ABB RobotStudio station: 101229220_Individual_Assignment_RSD.rspag

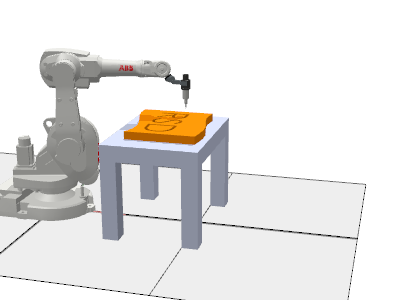
--- station ---
Station Project2 (saved by RobotStudio 24.1.10713.1)
Controller IRB1600_6_120
  mechanical unit ROB_1: IRB1600_6_120__02, 6 joints, base frame (0, 0, 0) mm
Layout (positions relative to the parent item):
  - IRB1600_6_120__02 [mechanism, from %ABB.RobotStudio.Models.IRB1600%\IRB1600_6_120_G_03.rslib] at (0, 0, 0) mm; joint values [0.2858, -0.0359, 0.0676, -0.2293, 0.9102, 0.378] (rad or m)
  - MyTool [mechanism, from Training Objects\myTool.rslib] at (742.97, 206.13, 890.95) mm, rotated rx -180 ry 38 rz 179.42 deg
  - Table [part] at (800, 0, 0) mm, rotated rx 0 ry 0 rz 90 deg, size 800 x 600 x 600 mm
  - RSD_Flag_3 [part] at (840.17, 31.01, 600) mm, rotated rx 0 ry 0 rz -90 deg, size 540.6 x 505.2 x 50 mm
Attachment: MyTool is attached to IRB1600_6_120__02 / Link6
Attachment: RSD_Flag_3 is attached to Table
Targets, tools, work objects and paths stored in the station and not in the controller backup, written as RAPID:
! task T_ROB1
MODULE Module1
  CONST robtarget Target_1090:=[[359.518,326.698,50],[0,0,1,0],[-1,0,-1,0],[9E+09,9E+09,9E+09,9E+09,9E+09,9E+09]];
  CONST robtarget Target_1100:=[[359.518,326.698,50],[0,0,1,0],[0,0,-1,0],[9E+09,9E+09,9E+09,9E+09,9E+09,9E+09]];
  CONST robtarget Target_1110:=[[359.518,326.698,50],[0,0,1,0],[0,0,-1,0],[9E+09,9E+09,9E+09,9E+09,9E+09,9E+09]];
  CONST robtarget Target_1120:=[[359.518,326.698,50],[0,0,1,0],[0,0,0,0],[9E+09,9E+09,9E+09,9E+09,9E+09,9E+09]];
  CONST robtarget Target_150_2:=[[193.305,628.255,70],[0,0,1,0],[0,0,0,0],[9E+09,9E+09,9E+09,9E+09,9E+09,9E+09]];
  CONST robtarget Target_310_2:=[[193.305,628.255,70],[0,0,1,0],[0,0,0,0],[9E+09,9E+09,9E+09,9E+09,9E+09,9E+09]];
  CONST robtarget Target_410_2:=[[359.518,611.634,70],[0,0,1,0],[0,0,0,0],[9E+09,9E+09,9E+09,9E+09,9E+09,9E+09]];
  CONST robtarget Target_930_2:=[[378.513525558,343.318900025,50],[0,0,1,0],[0,0,0,0],[9E+09,9E+09,9E+09,9E+09,9E+09,9E+09]];
  CONST robtarget Target_1130:=[[212.30091872,326.697639341,50],[0,1,0,0],[0,0,0,0],[9E+09,9E+09,9E+09,9E+09,9E+09,9E+09]];
  CONST robtarget Target_1140:=[[359.517799062,326.697639341,50],[0,1,0,0],[0,0,0,0],[9E+09,9E+09,9E+09,9E+09,9E+09,9E+09]];
  CONST robtarget Target_1150:=[[356.586817826,266.779478617,50],[0,-0.64587981,0.763439107,0],[0,0,0,0],[9E+09,9E+09,9E+09,9E+09,9E+09,9E+09]];
  CONST robtarget Target_1160:=[[347.459964861,240.920061884,50],[0,-0.495864219,0.868400067,0],[0,0,0,0],[9E+09,9E+09,9E+09,9E+09,9E+09,9E+09]];
  CONST robtarget Target_1170:=[[333.176068961,224.261700172,50],[0,-0.337129953,0.941458122,0],[0,0,0,0],[9E+09,9E+09,9E+09,9E+09,9E+09,9E+09]];
  CONST robtarget Target_1180:=[[313.586726012,213.020088593,50],[0,-0.178855224,0.983875403,0],[0,0,0,0],[9E+09,9E+09,9E+09,9E+09,9E+09,9E+09]];
  CONST robtarget Target_1190:=[[296.334747847,208.790571366,50],[0,-0.066549315,0.997783137,0],[0,0,0,0],[9E+09,9E+09,9E+09,9E+09,9E+09,9E+09]];
  CONST robtarget Target_1200:=[[265.874803603,209.643895017,50],[0,0.098590622,0.995128077,0],[0,0,0,0],[9E+09,9E+09,9E+09,9E+09,9E+09,9E+09]];
  CONST robtarget Target_1210:=[[245.580541116,217.101201708,50],[0,0.253457957,0.967346403,0],[0,0,0,0],[9E+09,9E+09,9E+09,9E+09,9E+09,9E+09]];
  CONST robtarget Target_1220:=[[229.552896885,230.049460588,50],[0,0.410722051,0.911760603,0],[0,0,0,0],[9E+09,9E+09,9E+09,9E+09,9E+09,9E+09]];
  CONST robtarget Target_1230:=[[221.019660374,242.663810214,50],[0,0.524154537,0.851623169,0],[0,0,0,0],[9E+09,9E+09,9E+09,9E+09,9E+09,9E+09]];
  CONST robtarget Target_1240:=[[214.155970136,266.853680674,50],[0,0.663168665,0.748469987,0],[0,0,0,0],[9E+09,9E+09,9E+09,9E+09,9E+09,9E+09]];
  CONST robtarget Target_1250:=[[212.30091872,326.697639341,50],[0,0.707106781,0.707106781,0],[0,0,0,0],[9E+09,9E+09,9E+09,9E+09,9E+09,9E+09]];
  CONST robtarget Target_1260:=[[297.781687951,611.633536777,50],[0,1,0,0],[0,0,0,0],[9E+09,9E+09,9E+09,9E+09,9E+09,9E+09]];
  CONST robtarget Target_1270:=[[359.517799062,611.633536777,50],[0,1,0,0],[0,0,0,0],[9E+09,9E+09,9E+09,9E+09,9E+09,9E+09]];
  CONST robtarget Target_1280:=[[297.781687951,611.633536777,50],[0,1,0,0],[0,0,0,0],[9E+09,9E+09,9E+09,9E+09,9E+09,9E+09]];
  CONST robtarget Target_120_2:=[[522.92,479.312,50],[0,-0.111729096,0.993738703,0],[0,0,-1,0],[9E+09,9E+09,9E+09,9E+09,9E+09,9E+09]];
  PROC Path_1()
    MoveL Target_140,v1500,fine,MyTool\WObj:=Table_Workobject;
    MoveL Target_130,v1500,fine,MyTool\WObj:=Table_Workobject;
    MoveC Target_120,Target_110,v1500,fine,MyTool\WObj:=Table_Workobject;
    MoveC Target_100,Target_90,v1500,fine,MyTool\WObj:=Table_Workobject;
    MoveL Target_80,v1500,fine,MyTool\WObj:=Table_Workobject;
    MoveC Target_70,Target_60,v1500,fine,MyTool\WObj:=Table_Workobject;
    MoveC Target_50,Target_40,v1500,fine,MyTool\WObj:=Table_Workobject;
    MoveC Target_30,Target_20,v1500,fine,MyTool\WObj:=Table_Workobject;
    MoveL Target_10,v1500,fine,MyTool\WObj:=Table_Workobject;
    MoveL Target_140_2,v1500,fine,MyTool\WObj:=Table_Workobject;
  ENDPROC
  PROC Path_2()
    MoveL Target_160,v1500,fine,MyTool\WObj:=Table_Workobject;
    MoveL Target_170,v1500,fine,MyTool\WObj:=Table_Workobject;
    MoveC Target_180,Target_190,v150,fine,MyTool\WObj:=Table_Workobject;
    MoveC Target_200,Target_210,v150,fine,MyTool\WObj:=Table_Workobject;
    MoveC Target_220,Target_230,v150,fine,MyTool\WObj:=Table_Workobject;
    MoveC Target_240,Target_250,v150,fine,MyTool\WObj:=Table_Workobject;
    MoveL Target_260,v1500,fine,MyTool\WObj:=Table_Workobject;
    MoveL Target_270,v1500,fine,MyTool\WObj:=Table_Workobject;
    MoveL Target_280,v1500,fine,MyTool\WObj:=Table_Workobject;
    MoveL Target_290,v1500,fine,MyTool\WObj:=Table_Workobject;
    MoveL Target_300,v1500,fine,MyTool\WObj:=Table_Workobject;
    MoveL Target_310,v1500,fine,MyTool\WObj:=Table_Workobject;
    MoveL Target_150,v1500,fine,MyTool\WObj:=Table_Workobject;
    MoveL Target_160,v1500,fine,MyTool\WObj:=Table_Workobject;
    MoveL Target_160_2,v1500,fine,MyTool\WObj:=Table_Workobject;
    MoveL Target_1290,v1000,z100,MyTool\WObj:=Table_Workobject;
    MoveL Target_400,v1500,fine,MyTool\WObj:=Table_Workobject;
    MoveC Target_390,Target_380,v150,fine,MyTool\WObj:=Table_Workobject;
    MoveC Target_370,Target_360,v150,fine,MyTool\WObj:=Table_Workobject;
    MoveC Target_350,Target_340,v150,fine,MyTool\WObj:=Table_Workobject;
    MoveL Target_330,v1500,fine,MyTool\WObj:=Table_Workobject;
    MoveL Target_1290,v1000,z100,MyTool\WObj:=Table_Workobject;
    MoveL Target_1290_2,v1000,z100,MyTool\WObj:=Table_Workobject;
  ENDPROC
  PROC Path_4()
    MoveL Target_930_2,v100,fine,MyTool\WObj:=Table_Workobject;
    MoveL Target_940,v600,fine,MyTool\WObj:=Table_Workobject;
    MoveL Target_950,v600,fine,MyTool\WObj:=Table_Workobject;
    MoveL Target_820,v600,fine,MyTool\WObj:=Table_Workobject;
    MoveC Target_830,Target_840,v600,fine,MyTool\WObj:=Table_Workobject;
    MoveC Target_850,Target_860,v600,fine,MyTool\WObj:=Table_Workobject;
    MoveC Target_870,Target_880,v600,fine,MyTool\WObj:=Table_Workobject;
    MoveC Target_890,Target_900,v600,fine,MyTool\WObj:=Table_Workobject;
    MoveL Target_910,v600,fine,MyTool\WObj:=Table_Workobject;
    MoveL Target_920,v600,fine,MyTool\WObj:=Table_Workobject;
    MoveL Target_930,v600,fine,MyTool\WObj:=Table_Workobject;
    MoveL Target_930_3,v600,fine,MyTool\WObj:=Table_Workobject;
    MoveL Target_1080,v600,fine,MyTool\WObj:=Table_Workobject;
    MoveL Target_1070,v600,fine,MyTool\WObj:=Table_Workobject;
    MoveC Target_1060,Target_1050,v600,fine,MyTool\WObj:=Table_Workobject;
    MoveC Target_1040,Target_1030,v600,fine,MyTool\WObj:=Table_Workobject;
    MoveC Target_1020,Target_1010,v600,fine,MyTool\WObj:=Table_Workobject;
    MoveC Target_1000,Target_990,v600,fine,MyTool\WObj:=Table_Workobject;
    MoveC Target_980,Target_970,v600,fine,MyTool\WObj:=Table_Workobject;
    MoveL Target_960,v600,fine,MyTool\WObj:=Table_Workobject;
  ENDPROC
  PROC Path_3()
    MoveL Target_520,v150,fine,MyTool\WObj:=Table_Workobject;
    MoveL Target_530,v150,fine,MyTool\WObj:=Table_Workobject;
    MoveL Target_540,v150,fine,MyTool\WObj:=Table_Workobject;
    MoveC Target_550,Target_560,v150,fine,MyTool\WObj:=Table_Workobject;
    MoveC Target_570,Target_580,v150,fine,MyTool\WObj:=Table_Workobject;
    MoveC Target_590,Target_600,v150,fine,MyTool\WObj:=Table_Workobject;
    MoveL Target_610,v150,fine,MyTool\WObj:=Table_Workobject;
    MoveC Target_620,Target_630,v150,fine,MyTool\WObj:=Table_Workobject;
    MoveC Target_640,Target_650,v150,fine,MyTool\WObj:=Table_Workobject;
    MoveC Target_660,Target_670,v150,fine,MyTool\WObj:=Table_Workobject;
    MoveC Target_680,Target_690,v150,fine,MyTool\WObj:=Table_Workobject;
    MoveL Target_700,v150,fine,MyTool\WObj:=Table_Workobject;
    MoveL Target_710,v150,fine,MyTool\WObj:=Table_Workobject;
    MoveL Target_720,v150,fine,MyTool\WObj:=Table_Workobject;
    MoveC Target_730,Target_740,v150,fine,MyTool\WObj:=Table_Workobject;
    MoveC Target_750,Target_760,v150,fine,MyTool\WObj:=Table_Workobject;
    MoveC Target_770,Target_780,v150,fine,MyTool\WObj:=Table_Workobject;
    MoveC Target_790,Target_800,v150,fine,MyTool\WObj:=Table_Workobject;
    MoveL Target_810,v150,fine,MyTool\WObj:=Table_Workobject;
    MoveL Target_420,v150,fine,MyTool\WObj:=Table_Workobject;
    MoveL Target_430,v150,fine,MyTool\WObj:=Table_Workobject;
    MoveC Target_440,Target_450,v150,fine,MyTool\WObj:=Table_Workobject;
    MoveC Target_460,Target_470,v150,fine,MyTool\WObj:=Table_Workobject;
    MoveC Target_480,Target_490,v150,fine,MyTool\WObj:=Table_Workobject;
    MoveC Target_500,Target_510,v150,fine,MyTool\WObj:=Table_Workobject;
    MoveL Target_520_2,v150,fine,MyTool\WObj:=Table_Workobject;
    MoveL Target_520_2_2,v150,fine,MyTool\WObj:=Table_Workobject;
  ENDPROC
ENDMODULE


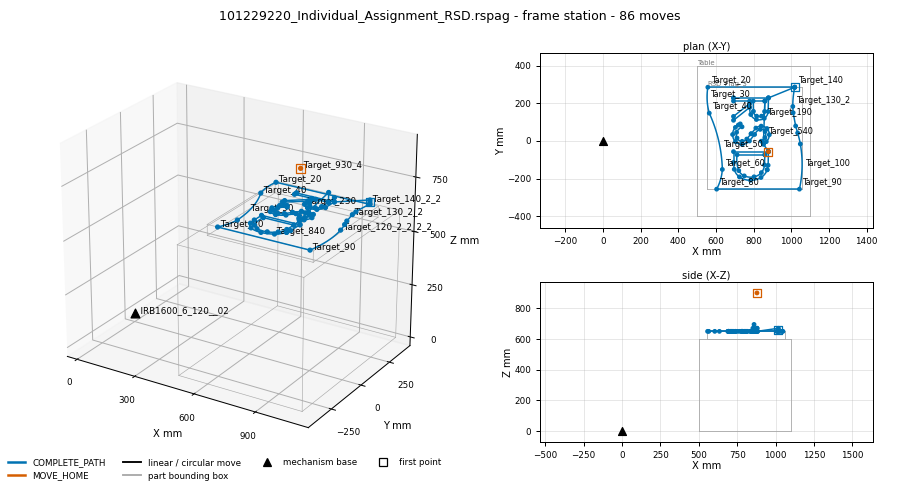
[picture p0: tool path of 101229220_Individual_Assignment_RSD.rspag in frame station, 86 of 86 moves have a stored position in this frame; points joined in program order, loops and branches not executed]
--- Controller Data/IRB1600_6_120/RAPID/TASK1/PROGMOD/CalibData.mod ---
MODULE CalibData
    PERS tooldata MyTool:=[TRUE,[[31.792631019,0,229.638935148],[0.945518576,0,0.325568154,0]],[1,[0,0,1],[1,0,0,0],0,0,0]];
    PERS wobjdata Table_Workobject:=[FALSE,TRUE,"",[[500,-400,600],[1,0,0,0]],[[0,0,0],[1,0,0,0]]];
ENDMODULE

--- Controller Data/IRB1600_6_120/RAPID/TASK1/PROGMOD/Module1.mod ---
MODULE Module1
        CONST robtarget Target_10:=[[517.947181876,684.868566444,50],[0,0,1,0],[0,0,0,0],[9E+09,9E+09,9E+09,9E+09,9E+09,9E+09]];
    CONST robtarget Target_20:=[[57.164143305,684.868566444,50],[0,0,1,0],[0,0,0,0],[9E+09,9E+09,9E+09,9E+09,9E+09,9E+09]];
    CONST robtarget Target_30:=[[53.433855577,615.547724999,50],[0,0.731366794,-0.68198432,0],[0,0,0,0],[9E+09,9E+09,9E+09,9E+09,9E+09,9E+09]];
    CONST robtarget Target_40:=[[64.693067941,547.312048631,50],[0,-0.11173174,0.993738405,0],[0,0,0,0],[9E+09,9E+09,9E+09,9E+09,9E+09,9E+09]];
    CONST robtarget Target_50:=[[124.654371405,349.660467509,50],[0,-0.11173174,0.993738405,0],[0,0,0,0],[9E+09,9E+09,9E+09,9E+09,9E+09,9E+09]];
    CONST robtarget Target_60:=[[134.028407273,248.711946133,50],[0,-0.11173174,0.993738405,0],[0,0,0,0],[9E+09,9E+09,9E+09,9E+09,9E+09,9E+09]];
    CONST robtarget Target_70:=[[125.076045967,197.014301808,50],[0,-0.11173174,0.993738405,0],[0,0,0,0],[9E+09,9E+09,9E+09,9E+09,9E+09,9E+09]];
    CONST robtarget Target_80:=[[103.797346016,144.237182321,50],[0,-0.11173174,0.993738405,0],[0,0,0,0],[9E+09,9E+09,9E+09,9E+09,9E+09,9E+09]];
    CONST robtarget Target_90:=[[542.968469011,144.237182321,50],[0,-0.11173174,0.993738405,0],[0,0,0,0],[9E+09,9E+09,9E+09,9E+09,9E+09,9E+09]];
    CONST robtarget Target_100:=[[556.357586504,247.055488013,50],[0,-0.11173174,0.993738405,0],[0,0,0,0],[9E+09,9E+09,9E+09,9E+09,9E+09,9E+09]];
    CONST robtarget Target_110:=[[555.000554572,348.782636867,50],[0,-0.11173174,0.993738405,0],[0,0,0,0],[9E+09,9E+09,9E+09,9E+09,9E+09,9E+09]];
    CONST robtarget Target_120:=[[509.880233717,547.312048631,50],[0,-0.11173174,0.993738405,0],[0,0,0,0],[9E+09,9E+09,9E+09,9E+09,9E+09,9E+09]];
    CONST robtarget Target_130:=[[508.670492721,615.825242702,50],[0,-0.11173174,0.993738405,0],[0,0,0,0],[9E+09,9E+09,9E+09,9E+09,9E+09,9E+09]];
    CONST robtarget Target_140:=[[517.947181876,684.868566444,50],[0,-0.11173174,0.993738405,0],[0,0,0,0],[9E+09,9E+09,9E+09,9E+09,9E+09,9E+09]];
    CONST robtarget Target_150:=[[193.305192225,628.254797461,50],[0,0,1,0],[0,0,0,0],[9E+09,9E+09,9E+09,9E+09,9E+09,9E+09]];
    CONST robtarget Target_160:=[[378.513525558,628.254797461,50],[0,0,1,0],[0,0,0,0],[9E+09,9E+09,9E+09,9E+09,9E+09,9E+09]];
    CONST robtarget Target_170:=[[377.103686482,555.981994309,50],[0,0,1,0],[0,0,0,0],[9E+09,9E+09,9E+09,9E+09,9E+09,9E+09]];
    CONST robtarget Target_180:=[[370.017390075,534.20369069,50],[0,0,1,0],[0,0,0,0],[9E+09,9E+09,9E+09,9E+09,9E+09,9E+09]];
    CONST robtarget Target_190:=[[356.475514741,519.845592733,50],[0,0,1,0],[0,0,0,0],[9E+09,9E+09,9E+09,9E+09,9E+09,9E+09]];
    CONST robtarget Target_200:=[[337.739495443,512.536690156,50],[0,0,1,0],[0,0,0,0],[9E+09,9E+09,9E+09,9E+09,9E+09,9E+09]];
    CONST robtarget Target_210:=[[314.699756861,513.723923062,50],[0,0,1,0],[0,0,0,0],[9E+09,9E+09,9E+09,9E+09,9E+09,9E+09]];
    CONST robtarget Target_220:=[[296.817061215,523.258887338,50],[0,0,1,0],[0,0,0,0],[9E+09,9E+09,9E+09,9E+09,9E+09,9E+09]];
    CONST robtarget Target_230:=[[284.796328042,540.102754192,50],[0,0,1,0],[0,0,0,0],[9E+09,9E+09,9E+09,9E+09,9E+09,9E+09]];
    CONST robtarget Target_240:=[[279.194072767,566.258979151,50],[0,0,1,0],[0,0,0,0],[9E+09,9E+09,9E+09,9E+09,9E+09,9E+09]];
    CONST robtarget Target_250:=[[278.785961455,577.574792787,50],[0,0,1,0],[0,0,0,0],[9E+09,9E+09,9E+09,9E+09,9E+09,9E+09]];
    CONST robtarget Target_260:=[[193.305192225,509.531506862,50],[0,0,1,0],[0,0,0,0],[9E+09,9E+09,9E+09,9E+09,9E+09,9E+09]];
    CONST robtarget Target_270:=[[193.305192225,530.085476547,50],[0,0,1,0],[0,0,0,0],[9E+09,9E+09,9E+09,9E+09,9E+09,9E+09]];
    CONST robtarget Target_280:=[[278.785961455,598.128762471,50],[0,0,1,0],[0,0,0,0],[9E+09,9E+09,9E+09,9E+09,9E+09,9E+09]];
    CONST robtarget Target_290:=[[278.785961455,611.633536777,50],[0,0,1,0],[0,0,0,0],[9E+09,9E+09,9E+09,9E+09,9E+09,9E+09]];
    CONST robtarget Target_300:=[[193.305192225,611.633536777,50],[0,0,1,0],[0,0,0,0],[9E+09,9E+09,9E+09,9E+09,9E+09,9E+09]];
    CONST robtarget Target_310:=[[193.305192225,628.254797461,50],[0,0,1,0],[0,0,0,0],[9E+09,9E+09,9E+09,9E+09,9E+09,9E+09]];
    CONST robtarget Target_320:=[[359.517799062,611.633536777,50],[0,0,1,0],[0,0,0,0],[9E+09,9E+09,9E+09,9E+09,9E+09,9E+09]];
    CONST robtarget Target_330:=[[297.781687951,611.633536777,50],[0,0,1,0],[0,0,0,0],[9E+09,9E+09,9E+09,9E+09,9E+09,9E+09]];
    CONST robtarget Target_340:=[[298.857617772,557.095025158,50],[0,0,1,0],[0,0,0,0],[9E+09,9E+09,9E+09,9E+09,9E+09,9E+09]];
    CONST robtarget Target_350:=[[305.461600812,540.13985522,50],[0,0,1,0],[0,0,0,0],[9E+09,9E+09,9E+09,9E+09,9E+09,9E+09]];
    CONST robtarget Target_360:=[[315.961191824,531.495315623,50],[0,0,1,0],[0,0,0,0],[9E+09,9E+09,9E+09,9E+09,9E+09,9E+09]];
    CONST robtarget Target_370:=[[329.02075379,528.527233358,50],[0,0,1,0],[0,0,0,0],[9E+09,9E+09,9E+09,9E+09,9E+09,9E+09]];
    CONST robtarget Target_380:=[[341.783507529,531.56951768,50],[0,0,1,0],[0,0,0,0],[9E+09,9E+09,9E+09,9E+09,9E+09,9E+09]];
    CONST robtarget Target_390:=[[352.023391343,540.102754192,50],[0,0,1,0],[0,0,0,0],[9E+09,9E+09,9E+09,9E+09,9E+09,9E+09]];
    CONST robtarget Target_400:=[[358.2563641,556.130398422,50],[0,0,1,0],[0,0,0,0],[9E+09,9E+09,9E+09,9E+09,9E+09,9E+09]];
    CONST robtarget Target_410:=[[359.517799062,611.633536777,50],[0,0,1,0],[0,0,0,0],[9E+09,9E+09,9E+09,9E+09,9E+09,9E+09]];
    CONST robtarget Target_420:=[[286.651379458,437.963623249,50],[0,0,1,0],[0,0,0,0],[9E+09,9E+09,9E+09,9E+09,9E+09,9E+09]];
    CONST robtarget Target_430:=[[311.842977681,468.312264408,50],[0,0,1,0],[0,0,0,0],[9E+09,9E+09,9E+09,9E+09,9E+09,9E+09]];
    CONST robtarget Target_440:=[[328.946551733,477.216511203,50],[0,0,1,0],[0,0,0,0],[9E+09,9E+09,9E+09,9E+09,9E+09,9E+09]];
    CONST robtarget Target_450:=[[340.039759199,478.663451307,50],[0,0,1,0],[0,0,0,0],[9E+09,9E+09,9E+09,9E+09,9E+09,9E+09]];
    CONST robtarget Target_460:=[[356.883626052,475.361459787,50],[0,0,1,0],[0,0,0,0],[9E+09,9E+09,9E+09,9E+09,9E+09,9E+09]];
    CONST robtarget Target_470:=[[370.833612697,465.715192426,50],[0,0,1,0],[0,0,0,0],[9E+09,9E+09,9E+09,9E+09,9E+09,9E+09]];
    CONST robtarget Target_480:=[[380.034667719,450.800579045,50],[0,0,1,0],[0,0,0,0],[9E+09,9E+09,9E+09,9E+09,9E+09,9E+09]];
    CONST robtarget Target_490:=[[383.262457182,433.029186483,50],[0,0,1,0],[0,0,0,0],[9E+09,9E+09,9E+09,9E+09,9E+09,9E+09]];
    CONST robtarget Target_500:=[[379.478152294,414.070561016,50],[0,0,1,0],[0,0,0,0],[9E+09,9E+09,9E+09,9E+09,9E+09,9E+09]];
    CONST robtarget Target_510:=[[367.04930781,396.262067426,50],[0,0,1,0],[0,0,0,0],[9E+09,9E+09,9E+09,9E+09,9E+09,9E+09]];
    CONST robtarget Target_520:=[[351.912088258,383.684818828,50],[0,0,1,0],[0,0,0,0],[9E+09,9E+09,9E+09,9E+09,9E+09,9E+09]];
    CONST robtarget Target_530:=[[340.522072567,398.710735295,50],[0,0,1,0],[0,0,0,0],[9E+09,9E+09,9E+09,9E+09,9E+09,9E+09]];
    CONST robtarget Target_540:=[[359.629102147,417.743562819,50],[0,0,1,0],[0,0,0,0],[9E+09,9E+09,9E+09,9E+09,9E+09,9E+09]];
    CONST robtarget Target_550:=[[364.266730686,434.884237899,50],[0,0,1,0],[0,0,0,0],[9E+09,9E+09,9E+09,9E+09,9E+09,9E+09]];
    CONST robtarget Target_560:=[[360.44532477,450.355366705,50],[0,0,1,0],[0,0,0,0],[9E+09,9E+09,9E+09,9E+09,9E+09,9E+09]];
    CONST robtarget Target_570:=[[349.945733758,460.150038179,50],[0,0,1,0],[0,0,0,0],[9E+09,9E+09,9E+09,9E+09,9E+09,9E+09]];
    CONST robtarget Target_580:=[[334.919817291,461.374372114,50],[0,0,1,0],[0,0,0,0],[9E+09,9E+09,9E+09,9E+09,9E+09,9E+09]];
    CONST robtarget Target_590:=[[323.270094402,455.73501581,50],[0,0,1,0],[0,0,0,0],[9E+09,9E+09,9E+09,9E+09,9E+09,9E+09]];
    CONST robtarget Target_600:=[[305.201893614,434.401924531,50],[0,0,1,0],[0,0,0,0],[9E+09,9E+09,9E+09,9E+09,9E+09,9E+09]];
    CONST robtarget Target_610:=[[277.672930606,399.823766144,50],[0,0,1,0],[0,0,0,0],[9E+09,9E+09,9E+09,9E+09,9E+09,9E+09]];
    CONST robtarget Target_620:=[[259.678931875,386.541598008,50],[0,0,1,0],[0,0,0,0],[9E+09,9E+09,9E+09,9E+09,9E+09,9E+09]];
    CONST robtarget Target_630:=[[238.67974985,381.310353016,50],[0,0,1,0],[0,0,0,0],[9E+09,9E+09,9E+09,9E+09,9E+09,9E+09]];
    CONST robtarget Target_640:=[[219.758225411,385.168859961,50],[0,0,1,0],[0,0,0,0],[9E+09,9E+09,9E+09,9E+09,9E+09,9E+09]];
    CONST robtarget Target_650:=[[203.470873982,396.744380794,50],[0,0,1,0],[0,0,0,0],[9E+09,9E+09,9E+09,9E+09,9E+09,9E+09]];
    CONST robtarget Target_660:=[[192.30346446,413.810853818,50],[0,0,1,0],[0,0,0,0],[9E+09,9E+09,9E+09,9E+09,9E+09,9E+09]];
    CONST robtarget Target_670:=[[188.556260601,434.216419389,50],[0,0,1,0],[0,0,0,0],[9E+09,9E+09,9E+09,9E+09,9E+09,9E+09]];
    CONST robtarget Target_680:=[[192.192161375,454.213873649,50],[0,0,1,0],[0,0,0,0],[9E+09,9E+09,9E+09,9E+09,9E+09,9E+09]];
    CONST robtarget Target_690:=[[203.322469869,471.799761069,50],[0,0,1,0],[0,0,0,0],[9E+09,9E+09,9E+09,9E+09,9E+09,9E+09]];
    CONST robtarget Target_700:=[[218.90490176,484.562514809,50],[0,0,1,0],[0,0,0,0],[9E+09,9E+09,9E+09,9E+09,9E+09,9E+09]];
    CONST robtarget Target_710:=[[229.033482489,490.535780367,50],[0,0,1,0],[0,0,0,0],[9E+09,9E+09,9E+09,9E+09,9E+09,9E+09]];
    CONST robtarget Target_720:=[[238.420042652,474.879146419,50],[0,0,1,0],[0,0,0,0],[9E+09,9E+09,9E+09,9E+09,9E+09,9E+09]];
    CONST robtarget Target_730:=[[219.609821298,460.929159774,50],[0,0,1,0],[0,0,0,0],[9E+09,9E+09,9E+09,9E+09,9E+09,9E+09]];
    CONST robtarget Target_740:=[[209.481240569,445.420929939,50],[0,0,1,0],[0,0,0,0],[9E+09,9E+09,9E+09,9E+09,9E+09,9E+09]];
    CONST robtarget Target_750:=[[207.551987097,434.216419389,50],[0,0,1,0],[0,0,0,0],[9E+09,9E+09,9E+09,9E+09,9E+09,9E+09]];
    CONST robtarget Target_760:=[[211.855706381,415.665905233,50],[0,0,1,0],[0,0,0,0],[9E+09,9E+09,9E+09,9E+09,9E+09,9E+09]];
    CONST robtarget Target_770:=[[223.468328242,402.457939154,50],[0,0,1,0],[0,0,0,0],[9E+09,9E+09,9E+09,9E+09,9E+09,9E+09]];
    CONST robtarget Target_780:=[[238.939457048,397.9316137,50],[0,0,1,0],[0,0,0,0],[9E+09,9E+09,9E+09,9E+09,9E+09,9E+09]];
    CONST robtarget Target_790:=[[248.14051207,399.601159974,50],[0,0,1,0],[0,0,0,0],[9E+09,9E+09,9E+09,9E+09,9E+09,9E+09]];
    CONST robtarget Target_800:=[[263.574539848,410.063649958,50],[0,0,1,0],[0,0,0,0],[9E+09,9E+09,9E+09,9E+09,9E+09,9E+09]];
    CONST robtarget Target_810:=[[286.651379458,437.963623249,50],[0,0,1,0],[0,0,0,0],[9E+09,9E+09,9E+09,9E+09,9E+09,9E+09]];
    CONST robtarget Target_820:=[[371.835340462,247.15303464,50],[0,0,1,0],[0,0,0,0],[9E+09,9E+09,9E+09,9E+09,9E+09,9E+09]];
    CONST robtarget Target_830:=[[358.961283638,223.779386804,50],[0,0,1,0],[0,0,0,0],[9E+09,9E+09,9E+09,9E+09,9E+09,9E+09]];
    CONST robtarget Target_840:=[[339.112233491,206.156398356,50],[0,0,1,0],[0,0,0,0],[9E+09,9E+09,9E+09,9E+09,9E+09,9E+09]];
    CONST robtarget Target_850:=[[313.586726012,195.06319089,50],[0,0,1,0],[0,0,0,0],[9E+09,9E+09,9E+09,9E+09,9E+09,9E+09]];
    CONST robtarget Target_860:=[[283.571994108,191.353088059,50],[0,0,1,0],[0,0,0,0],[9E+09,9E+09,9E+09,9E+09,9E+09,9E+09]];
    CONST robtarget Target_870:=[[251.405402561,195.916514541,50],[0,0,1,0],[0,0,0,0],[9E+09,9E+09,9E+09,9E+09,9E+09,9E+09]];
    CONST robtarget Target_880:=[[224.729763205,209.34708679,50],[0,0,1,0],[0,0,0,0],[9E+09,9E+09,9E+09,9E+09,9E+09,9E+09]];
    CONST robtarget Target_890:=[[206.067945964,228.936429739,50],[0,0,1,0],[0,0,0,0],[9E+09,9E+09,9E+09,9E+09,9E+09,9E+09]];
    CONST robtarget Target_900:=[[197.237901226,249.638803537,50],[0,0,1,0],[0,0,0,0],[9E+09,9E+09,9E+09,9E+09,9E+09,9E+09]];
    CONST robtarget Target_910:=[[193.305192225,285.923609226,50],[0,0,1,0],[0,0,0,0],[9E+09,9E+09,9E+09,9E+09,9E+09,9E+09]];
    CONST robtarget Target_920:=[[193.305192225,343.318900025,50],[0,0,1,0],[0,0,0,0],[9E+09,9E+09,9E+09,9E+09,9E+09,9E+09]];
    CONST robtarget Target_930:=[[378.513525558,343.318900025,50],[0,0,1,0],[0,0,0,0],[9E+09,9E+09,9E+09,9E+09,9E+09,9E+09]];
    CONST robtarget Target_940:=[[376.843979284,270.971894817,50],[0,0,1,0],[0,0,0,0],[9E+09,9E+09,9E+09,9E+09,9E+09,9E+09]];
    CONST robtarget Target_950:=[[371.835340462,247.15303464,50],[0,0,1,0],[0,0,0,0],[9E+09,9E+09,9E+09,9E+09,9E+09,9E+09]];
    CONST robtarget Target_960:=[[359.517799062,326.697639341,50],[0,0,1,0],[0,0,0,0],[9E+09,9E+09,9E+09,9E+09,9E+09,9E+09]];
    CONST robtarget Target_970:=[[212.30091872,326.697639341,50],[0,0,1,0],[0,0,0,0],[9E+09,9E+09,9E+09,9E+09,9E+09,9E+09]];
    CONST robtarget Target_980:=[[214.155970136,266.853680674,50],[0,0,1,0],[0,0,0,0],[9E+09,9E+09,9E+09,9E+09,9E+09,9E+09]];
    CONST robtarget Target_990:=[[221.019660374,242.663810214,50],[0,0,1,0],[0,0,0,0],[9E+09,9E+09,9E+09,9E+09,9E+09,9E+09]];
    CONST robtarget Target_1000:=[[233.077494575,226.376458786,50],[0,0,1,0],[0,0,0,0],[9E+09,9E+09,9E+09,9E+09,9E+09,9E+09]];
    CONST robtarget Target_1010:=[[250.292371712,214.689634867,50],[0,0,1,0],[0,0,0,0],[9E+09,9E+09,9E+09,9E+09,9E+09,9E+09]];
    CONST robtarget Target_1020:=[[271.551260935,208.716369309,50],[0,0,1,0],[0,0,0,0],[9E+09,9E+09,9E+09,9E+09,9E+09,9E+09]];
    CONST robtarget Target_1030:=[[302.308013405,209.79229913,50],[0,0,1,0],[0,0,0,0],[9E+09,9E+09,9E+09,9E+09,9E+09,9E+09]];
    CONST robtarget Target_1040:=[[323.900811883,217.843222274,50],[0,0,1,0],[0,0,0,0],[9E+09,9E+09,9E+09,9E+09,9E+09,9E+09]];
    CONST robtarget Target_1050:=[[341.041486963,231.978714061,50],[0,0,1,0],[0,0,0,0],[9E+09,9E+09,9E+09,9E+09,9E+09,9E+09]];
    CONST robtarget Target_1060:=[[350.131238899,245.891599678,50],[0,0,1,0],[0,0,0,0],[9E+09,9E+09,9E+09,9E+09,9E+09,9E+09]];
    CONST robtarget Target_1070:=[[357.477242505,272.86404726,50],[0,0,1,0],[0,0,0,0],[9E+09,9E+09,9E+09,9E+09,9E+09,9E+09]];
    CONST robtarget Target_1080:=[[359.517799062,326.697639341,50],[0,0,1,0],[0,0,0,0],[9E+09,9E+09,9E+09,9E+09,9E+09,9E+09]];
    CONST robtarget Target_666:=[[183.88,401.02,106.66],[0.00241711,0.0181139,-0.998756,-0.0463868],[-1,0,-1,0],[9E+9,9E+9,9E+9,9E+9,9E+9,9E+9]];
     CONST robtarget Target_222:=[[354.00,267.59,54.80],[7.2429E-7,-0.313489,0.949592,-1.52255E-7],[-1,0,-1,0],[9E+9,9E+9,9E+9,9E+9,9E+9,9E+9]];
    CONST robtarget Target_140_2_2:=[[517.947,684.869,60],[0,-0.111729096,0.993738703,0],[0,0,0,0],[9E+09,9E+09,9E+09,9E+09,9E+09,9E+09]];
    CONST robtarget Target_130_2:=[[507.67,582.825,50],[0,-0.111729096,0.993738703,0],[0,0,0,0],[9E+09,9E+09,9E+09,9E+09,9E+09,9E+09]];
    CONST robtarget Target_130_2_2:=[[509.615,549.64,50],[0,-0.111729096,0.993738703,0],[0,0,-1,0],[9E+09,9E+09,9E+09,9E+09,9E+09,9E+09]];
    CONST robtarget Target_130_2_2_2:=[[522.92,479.31,50],[0,-0.111729096,0.993738703,0],[0,0,-1,0],[9E+09,9E+09,9E+09,9E+09,9E+09,9E+09]];
    CONST robtarget Target_120_2_2:=[[533.4,442.312,50],[0,-0.111729096,0.993738703,0],[0,0,-1,0],[9E+09,9E+09,9E+09,9E+09,9E+09,9E+09]];
    CONST robtarget Target_120_2_2_2:=[[540.1,418.312,50],[0,-0.111729096,0.993738703,0],[-1,0,-1,0],[9E+09,9E+09,9E+09,9E+09,9E+09,9E+09]];
    CONST robtarget Target_120_2_2_2_2:=[[547.57917033,383.940929313,50],[0,-0.111728012,0.993738824,0],[-1,0,-1,0],[9E+09,9E+09,9E+09,9E+09,9E+09,9E+09]];
    CONST robtarget Target_140_2:=[[517.947,684.869,70],[0,-0.111729096,0.993738703,0],[0,0,0,0],[9E+09,9E+09,9E+09,9E+09,9E+09,9E+09]];
    CONST robtarget Target_160_2:=[[378.514,628.255,70],[0,0,1,0],[0,0,0,0],[9E+09,9E+09,9E+09,9E+09,9E+09,9E+09]];
    CONST robtarget Target_1290:=[[359.517799062,611.633536777,50],[0,0.005199113,0.999986485,0],[0,0,0,0],[9E+09,9E+09,9E+09,9E+09,9E+09,9E+09]];
    CONST robtarget Target_1290_2:=[[359.518,611.634,95],[0,0.005201058,0.999986474,0],[0,0,0,0],[9E+09,9E+09,9E+09,9E+09,9E+09,9E+09]];
    CONST robtarget Target_520_2:=[[351.912088258,383.684818828,50],[0,0,1,0],[0,0,0,0],[9E+09,9E+09,9E+09,9E+09,9E+09,9E+09]];
    CONST robtarget Target_520_2_2:=[[351.912,383.685,70],[0,0,1,0],[0,0,0,0],[9E+09,9E+09,9E+09,9E+09,9E+09,9E+09]];
    CONST robtarget Target_930_2_2:=[[378.514,343.319,70],[0,0,1,0],[0,0,0,0],[9E+09,9E+09,9E+09,9E+09,9E+09,9E+09]];
    CONST robtarget Target_930_3:=[[378.514,343.319,70],[0,0,1,0],[0,0,0,0],[9E+09,9E+09,9E+09,9E+09,9E+09,9E+09]];
    CONST robtarget Target_930_4:=[[378.514,343.319,300],[0,0,1,0],[0,0,0,0],[9E+09,9E+09,9E+09,9E+09,9E+09,9E+09]];
!***********************************************************
    !
    ! Module:  Module1
    !
    ! Description:
    !   <Insert description here>
    !
    ! Author: Abdulswamad Rama Salim
    !
    ! Version: 1.0
    !
    !********************************4***************************


    !***********************************************************
    !
    ! Procedure main
    !
    !   This is the entry point of your program
    !
    !***********************************************************
    PROC main()
        !Add your code here
        COMPLETE_PATH;
        MOVE_HOME;
    ENDPROC
    PROC COMPLETE_PATH()
        WaitTime 2;
        MoveL Target_140_2_2,v150,fine,MyTool\WObj:=Table_Workobject;
        MoveL Target_140,v150,fine,MyTool\WObj:=Table_Workobject;
        MoveC Target_130,Target_130_2,v200,fine,MyTool\WObj:=Table_Workobject;
        MoveL Target_130_2_2,v150,z100,MyTool\WObj:=Table_Workobject;
        MoveL Target_130_2_2_2,v150,z100,MyTool\WObj:=Table_Workobject;
        MoveL Target_120_2_2,v150,z100,MyTool\WObj:=Table_Workobject;
        MoveC Target_120_2_2_2,Target_120_2_2_2_2,v150,z100,MyTool\WObj:=Table_Workobject;
        MoveC Target_100,Target_90,v150,fine,MyTool\WObj:=Table_Workobject;
        MoveL Target_80,v200,fine,MyTool\WObj:=Table_Workobject;
        MoveC Target_70,Target_60,v200,fine,MyTool\WObj:=Table_Workobject;
        MoveC Target_50,Target_40,v200,fine,MyTool\WObj:=Table_Workobject;
        MoveC Target_30,Target_20,v150,fine,MyTool\WObj:=Table_Workobject;
        MoveL Target_10,v150,fine,MyTool\WObj:=Table_Workobject;
        MoveL Target_140_2,v100,fine,MyTool\WObj:=Table_Workobject;
        MoveL Target_160,v150,fine,MyTool\WObj:=Table_Workobject;
        MoveL Target_170,v150,fine,MyTool\WObj:=Table_Workobject;
        MoveC Target_180,Target_190,v150,fine,MyTool\WObj:=Table_Workobject;
        MoveC Target_200,Target_210,v150,fine,MyTool\WObj:=Table_Workobject;
        MoveC Target_220,Target_230,v150,fine,MyTool\WObj:=Table_Workobject;
        MoveC Target_240,Target_250,v150,fine,MyTool\WObj:=Table_Workobject;
        MoveL Target_260,v150,fine,MyTool\WObj:=Table_Workobject;
        MoveL Target_270,v150,fine,MyTool\WObj:=Table_Workobject;
        MoveL Target_280,v300,fine,MyTool\WObj:=Table_Workobject;
        MoveL Target_290,v300,fine,MyTool\WObj:=Table_Workobject;
        MoveL Target_300,v300,fine,MyTool\WObj:=Table_Workobject;
        MoveL Target_310,v300,fine,MyTool\WObj:=Table_Workobject;
        MoveL Target_150,v1500,fine,MyTool\WObj:=Table_Workobject;
        MoveL Target_160,v150,fine,MyTool\WObj:=Table_Workobject;
        MoveL Target_160_2,v150,fine,MyTool\WObj:=Table_Workobject;
        MoveL Target_1290,v150,z100,MyTool\WObj:=Table_Workobject;
        MoveL Target_400,v150,fine,MyTool\WObj:=Table_Workobject;
        MoveC Target_390,Target_380,v150,fine,MyTool\WObj:=Table_Workobject;
        MoveC Target_370,Target_360,v150,fine,MyTool\WObj:=Table_Workobject;
        MoveC Target_350,Target_340,v150,fine,MyTool\WObj:=Table_Workobject;
        MoveL Target_330,v150,fine,MyTool\WObj:=Table_Workobject;
        MoveL Target_1290,v150,z100,MyTool\WObj:=Table_Workobject;
        MoveL Target_1290_2,v150,z100,MyTool\WObj:=Table_Workobject;
        MoveL Target_520,v150,fine,MyTool\WObj:=Table_Workobject;
        MoveL Target_530,v500,fine,MyTool\WObj:=Table_Workobject;
        MoveL Target_540,v500,fine,MyTool\WObj:=Table_Workobject;
        MoveC Target_550,Target_560,v150,fine,MyTool\WObj:=Table_Workobject;
        MoveC Target_570,Target_580,v150,fine,MyTool\WObj:=Table_Workobject;
        MoveC Target_590,Target_600,v150,fine,MyTool\WObj:=Table_Workobject;
        MoveL Target_610,v500,fine,MyTool\WObj:=Table_Workobject;
        MoveC Target_620,Target_630,v150,fine,MyTool\WObj:=Table_Workobject;
        MoveC Target_640,Target_650,v150,fine,MyTool\WObj:=Table_Workobject;
        MoveC Target_660,Target_670,v150,fine,MyTool\WObj:=Table_Workobject;
        MoveC Target_680,Target_690,v150,fine,MyTool\WObj:=Table_Workobject;
        MoveL Target_700,v200,fine,MyTool\WObj:=Table_Workobject;
        MoveL Target_710,v200,fine,MyTool\WObj:=Table_Workobject;
        MoveL Target_720,v200,fine,MyTool\WObj:=Table_Workobject;
        MoveC Target_730,Target_740,v150,fine,MyTool\WObj:=Table_Workobject;
        MoveC Target_750,Target_760,v150,fine,MyTool\WObj:=Table_Workobject;
        MoveC Target_770,Target_780,v150,fine,MyTool\WObj:=Table_Workobject;
        MoveC Target_790,Target_800,v150,fine,MyTool\WObj:=Table_Workobject;
        MoveL Target_810,v150,fine,MyTool\WObj:=Table_Workobject;
        MoveL Target_420,v150,fine,MyTool\WObj:=Table_Workobject;
        MoveL Target_430,v150,fine,MyTool\WObj:=Table_Workobject;
        MoveC Target_440,Target_450,v150,fine,MyTool\WObj:=Table_Workobject;
        MoveC Target_460,Target_470,v150,fine,MyTool\WObj:=Table_Workobject;
        MoveC Target_480,Target_490,v150,fine,MyTool\WObj:=Table_Workobject;
        MoveC Target_500,Target_510,v150,fine,MyTool\WObj:=Table_Workobject;
        MoveL Target_520_2,v150,fine,MyTool\WObj:=Table_Workobject;
        MoveL Target_520_2_2,v150,fine,MyTool\WObj:=Table_Workobject;
        MoveL Target_930_2_2,v50,fine,MyTool\WObj:=Table_Workobject;
        MoveL Target_930,v100,z100,MyTool\WObj:=Table_Workobject;
        MoveL Target_940,v150,fine,MyTool\WObj:=Table_Workobject;
        MoveL Target_950,v200,fine,MyTool\WObj:=Table_Workobject;
        MoveL Target_820,v150,fine,MyTool\WObj:=Table_Workobject;
        MoveC Target_830,Target_840,v150,fine,MyTool\WObj:=Table_Workobject;
        MoveC Target_850,Target_860,v150,fine,MyTool\WObj:=Table_Workobject;
        MoveC Target_870,Target_880,v150,fine,MyTool\WObj:=Table_Workobject;
        MoveC Target_890,Target_900,v150,fine,MyTool\WObj:=Table_Workobject;
        MoveL Target_910,v200,fine,MyTool\WObj:=Table_Workobject;
        MoveL Target_920,v200,fine,MyTool\WObj:=Table_Workobject;
        MoveL Target_930,v150,fine,MyTool\WObj:=Table_Workobject;
        MoveL Target_930_3,v600,fine,MyTool\WObj:=Table_Workobject;
        MoveL Target_1080,v200,fine,MyTool\WObj:=Table_Workobject;
        MoveL Target_1070,v200,fine,MyTool\WObj:=Table_Workobject;
        MoveC Target_1060,Target_1050,v150,fine,MyTool\WObj:=Table_Workobject;
        MoveC Target_1040,Target_1030,v150,fine,MyTool\WObj:=Table_Workobject;
        MoveC Target_1020,Target_1010,v150,fine,MyTool\WObj:=Table_Workobject;
        MoveC Target_1000,Target_990,v150,fine,MyTool\WObj:=Table_Workobject;
        MoveC Target_980,Target_970,v150,fine,MyTool\WObj:=Table_Workobject;
        MoveL Target_960,v200,fine,MyTool\WObj:=Table_Workobject;
    ENDPROC
    PROC MOVE_HOME()
        MoveL Target_930_4,v600,fine,MyTool\WObj:=Table_Workobject;
        WaitTime 2;
    ENDPROC
ENDMODULE
